{attribute 'qualified_only'}
{attribute 'strict'}
TYPE E_STATES :
(
	INIT := 0, // INIT 
	NOT_SAFE ,// NOT OK to move in the same state
	READY, // Safe to Move STATE
	OVERRIDE,
	SETUP
	
);
END_TYPE

(* stored: Version 1.1.0.1, ProductVersion 3.1.4024.3
   EnumerationTextList E_STATES: Id {5a8eaf0e-b91c-478f-882b-ab2b2b8d0678} *)
